{attribute addProperty BoxType "EL6201-0000-0017"}
{attribute addProperty Id "Slave_21A_DO0BIT10.125161Slave_21A_DO1BIT10.125162Slave_21A_DO2BIT10.125163Slave_21A_DO3BIT10.125164Slave_21B_DO0BIT10.125165Slave_21B_DO1BIT10.125166Slave_21B_DO2BIT10.125167Slave_21B_DO3BIT10.125168"}
{attribute addProperty CRC "607850430"}
{attribute addProperty SizeInBites "8"}
{attribute addProperty SizeInBytes "1"}
TYPE Slave_21_Outputs_243B0FBE :
STRUCT
	{attribute addProperty Name "Slave_21A_DO0"}
	Slave_21A_DO0 : BIT;
	{attribute addProperty Name "Slave_21A_DO1"}
	Slave_21A_DO1 : BIT;
	{attribute addProperty Name "Slave_21A_DO2"}
	Slave_21A_DO2 : BIT;
	{attribute addProperty Name "Slave_21A_DO3"}
	Slave_21A_DO3 : BIT;
	{attribute addProperty Name "Slave_21B_DO0"}
	Slave_21B_DO0 : BIT;
	{attribute addProperty Name "Slave_21B_DO1"}
	Slave_21B_DO1 : BIT;
	{attribute addProperty Name "Slave_21B_DO2"}
	Slave_21B_DO2 : BIT;
	{attribute addProperty Name "Slave_21B_DO3"}
	Slave_21B_DO3 : BIT;
END_STRUCT
END_TYPE

(* stored: Version 1.2.0.0, ProductVersion 3.1.4024.9
   DUT Slave_21_Outputs_243B0FBE: Id {989fc48a-cac4-4cfc-b1ab-f50eabd1cbaa} *)
